FUNCTION_BLOCK XtsAxisControl
VAR_INPUT
END_VAR
VAR_OUTPUT
END_VAR
VAR

	Axis					: AXIS_REF;
	
	BusyMoving				: BOOL;
	BusyStopping			: BOOL;
	Error					: BOOL;
	ErrorID					: UDINT;
	ErrorIDPrevious			: UDINT;
	ErrorStop				: BOOL;
	Disabled				: BOOL;
	Stopping				: BOOL;
	StandStill				: BOOL;
	DiscreteMotion			: BOOL;
	ContinuousMotion		: BOOL;
	SynchronizedMotion		: BOOL;
	Homing					: BOOL;
	ConstantVelocity		: BOOL;
	Accelerating			: BOOL;
	Decelerating			: BOOL;
	Status					: ST_AxisStatus;
	ErrorCount				: UINT;
	
	ErrorCountTrigger		: R_TRIG;
	
	Enable					: MC_Power;
	Restart					: MC_Reset;
	ReadStatus				: MC_ReadStatus;	
	MoveAbs1				: MC_MoveAbsolute;
	MoveAbs2				: MC_MoveAbsolute;
	MoveRel1				: MC_MoveRelative;
	MoveRel2				: MC_MoveRelative;
	MoveVel1				: MC_MoveVelocity;
	MoveVel2				: MC_MoveVelocity;
	StopWeak				: MC_Halt;
	StopStrong				: MC_Stop;
	
	MoveAbsCA				: MC_MoveAbsoluteCA;
	MoveRelCA				: MC_MoveRelativeCA;
	StopWeakCA				: MC_HaltCA;
	
END_VAR

// NETWORK 1

METHOD AutoErrorCheckAndReset : BOOL
VAR_INPUT
END_VAR

// Automatically check for errors on the NC axis, then reset them
// Use with caution, this could cause damage to a physical system if implemented without care

ReadStatus(Axis := Axis);
Restart(Axis := Axis);
ErrorCountTrigger(CLK := Error);

IF ErrorCountTrigger.Q THEN
	ErrorCount := ErrorCount + 1;
END_IF

IF Error THEN
	Restart.Execute := TRUE;
	IF Restart.Done THEN
		Restart.Execute := FALSE;
		AutoErrorCheckAndReset := TRUE;
	END_IF
END_IF
END_METHOD

PROPERTY AxisRef : AXIS_REF
GET
AxisRef := Axis;
END_GET
SET
END_SET
END_PROPERTY

METHOD CheckForErrors : BOOL
VAR_INPUT	
END_VAR

// Check for errors on the NC axis

ReadStatus(Axis := Axis);
ErrorCountTrigger(CLK := Error);

IF ErrorCountTrigger.Q THEN
	ErrorCount := ErrorCount + 1;
END_IF

IF Error THEN
	CheckForErrors := TRUE;
END_IF
END_METHOD

METHOD CyclicUpdate : BOOL
VAR_INPUT	
END_VAR
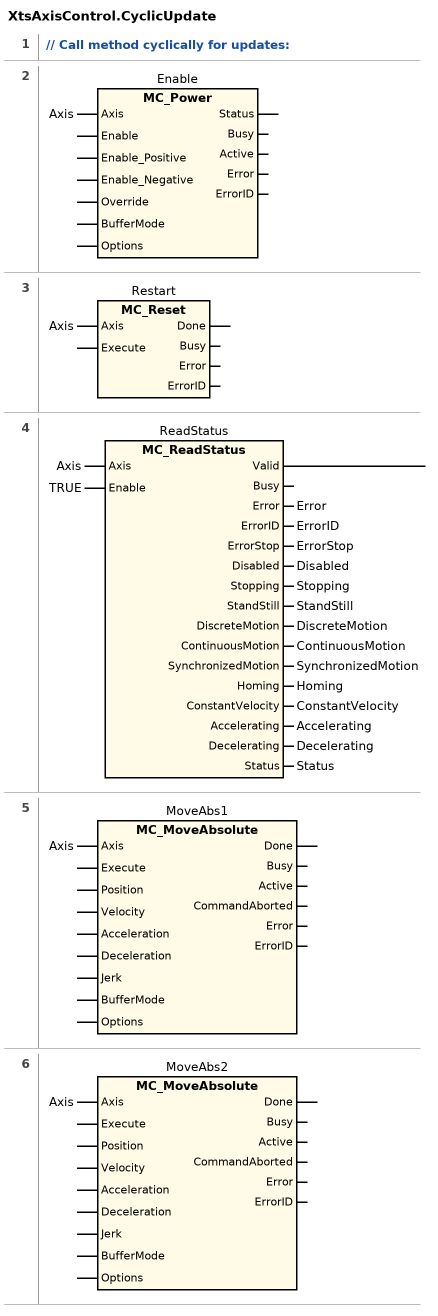
// NETWORK 1
// label: // Call method cyclically for updates

// NETWORK 2
Enable(Axis := Axis); // MC_Power

// NETWORK 3
Restart(Axis := Axis); // MC_Reset

// NETWORK 4
ReadStatus(
    Axis := Axis,
    Enable := TRUE,
    Error => Error,
    ErrorID => ErrorID,
    ErrorStop => ErrorStop,
    Disabled => Disabled,
    Stopping => Stopping,
    StandStill => StandStill,
    DiscreteMotion => DiscreteMotion,
    ContinuousMotion => ContinuousMotion,
    SynchronizedMotion => SynchronizedMotion,
    Homing => Homing,
    ConstantVelocity => ConstantVelocity,
    Accelerating => Accelerating,
    Decelerating => Decelerating,
    Status => Status); // MC_ReadStatus

// NETWORK 5
MoveAbs1(Axis := Axis); // MC_MoveAbsolute

// NETWORK 6
MoveAbs2(Axis := Axis); // MC_MoveAbsolute

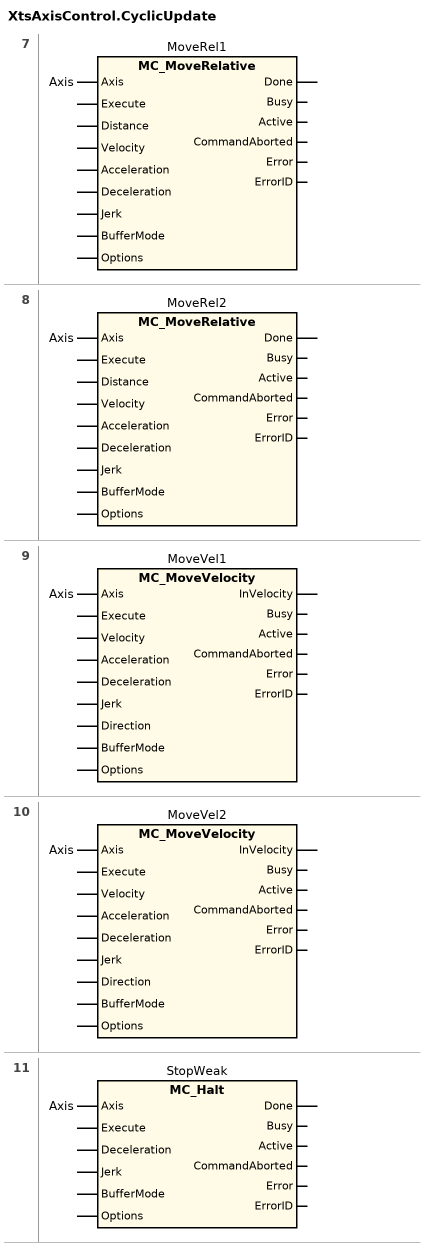
// NETWORK 7
MoveRel1(Axis := Axis); // MC_MoveRelative

// NETWORK 8
MoveRel2(Axis := Axis); // MC_MoveRelative

// NETWORK 9
MoveVel1(Axis := Axis); // MC_MoveVelocity

// NETWORK 10
MoveVel2(Axis := Axis); // MC_MoveVelocity

// NETWORK 11
StopWeak(Axis := Axis); // MC_Halt

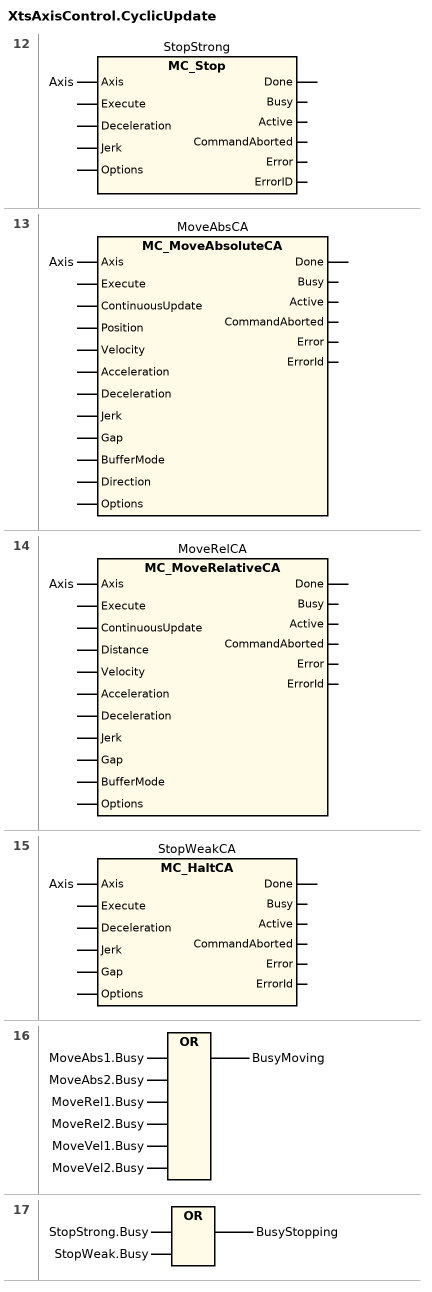
// NETWORK 12
StopStrong(Axis := Axis); // MC_Stop

// NETWORK 13
MoveAbsCA(Axis := Axis); // MC_MoveAbsoluteCA

// NETWORK 14
MoveRelCA(Axis := Axis); // MC_MoveRelativeCA

// NETWORK 15
StopWeakCA(Axis := Axis); // MC_HaltCA

// NETWORK 16
BusyMoving := MoveAbs1.Busy OR MoveAbs2.Busy OR MoveRel1.Busy OR MoveRel2.Busy OR MoveVel1.Busy OR MoveVel2.Busy;

// NETWORK 17
BusyStopping := StopStrong.Busy OR StopWeak.Busy;

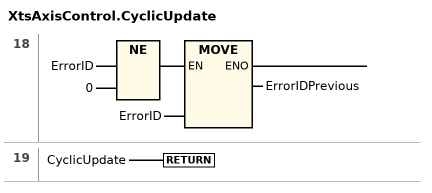
// NETWORK 18
IF ErrorID <> 0 THEN ErrorIDPrevious := ErrorID; END_IF

// NETWORK 19
IF CyclicUpdate THEN RETURN; END_IF
END_METHOD

METHOD MoveToPositionCA : BOOL
VAR_INPUT
	Position			: LREAL;
	Velocity			: LREAL;
	Options				: ST_MoveAbsoluteCAOptions;
END_VAR
MoveAbsCA(Axis := Axis);

MoveAbsCA.Position 			:= Position;
MoveAbsCA.Velocity 			:= Velocity;
MoveAbsCA.Direction			:= mcDirectionShortestWay;
MoveAbsCA.BufferMode		:= mcAborting;
MoveAbsCA.Options			:= Options;

MoveAbsCA.Execute 			:= TRUE;

IF MoveAbsCA.Done THEN
	MoveAbsCA.Execute := FALSE;
	MoveToPositionCA := TRUE;
END_IF
END_METHOD

METHOD PowerOff : BOOL
VAR_INPUT
END_VAR

// Disable the axis

Enable(Axis := Axis);

Enable.Enable 				:= FALSE;
Enable.Enable_Negative 		:= FALSE;
Enable.Enable_Positive 		:= FALSE;
Enable.Override 			:= 0;

IF NOT Enable.Status THEN
	PowerOff := TRUE;
END_IF
END_METHOD

METHOD PowerOn : BOOL
VAR_INPUT
END_VAR

// Enable the axis

Enable(Axis := Axis);

Enable.Enable 				:= TRUE;
Enable.Enable_Negative 		:= TRUE;
Enable.Enable_Positive 		:= TRUE;
Enable.Override 			:= 100;

IF Enable.Status THEN
	PowerOn := TRUE;
END_IF
END_METHOD

METHOD Reset : BOOL
VAR_INPUT
END_VAR

// Reset errors on the NC axis

Restart(Axis := Axis);

Restart.Execute 			:= TRUE;

IF Restart.Done THEN
	Restart.Execute := FALSE;
	Reset := TRUE;
END_IF
END_METHOD

END_FUNCTION_BLOCK

(* stored: Version 1.1.0.1, ProductVersion 3.1.4024.12
   POU XtsAxisControl: Id {ec1eec99-a289-419f-92b9-8b98742473d8}, SpecialFunc None
   Folder Movements: Id {e983c8f8-8927-4dc9-9aed-b49726e466f0}
   Folder Movements CA: Id {d9b65ed1-50f0-4c83-93a0-12db3bb625a2}
   Folder Power and Utility: Id {27299485-0fb2-48d8-a5a9-eb5b18706a1b}
   Method AutoErrorCheckAndReset: Id {c4558794-dce0-4723-8ae5-ffe53ab7450c}
   Property AxisRef: Id {3d5430da-c49f-45c9-9c96-126df32a8d8d}
   Get Get: Id {1cf6b178-fc4c-4283-8e80-0207ad4a2955}
   Set Set: Id {2f49716e-2bf5-4438-86ff-c3c2ebefa7b0}
   Method CheckForErrors: Id {1156e6bc-6693-4a8a-8e9b-2040f7a304f7}
   Method CyclicUpdate: Id {c275bfeb-5ff7-446d-85fb-f8549f5a0176}
   Method MoveToPositionCA: Id {be2b9eb0-de2c-483b-baa5-ac136c73c00c}
   Method PowerOff: Id {931cb592-80ae-4fd4-9bc7-23c7456ec9bf}
   Method PowerOn: Id {055fc17f-11ee-4864-95b6-aec8c64cb3a6}
   Method Reset: Id {42cec210-5b3f-4f2e-9099-2c39c8e00b0b} *)
